FUNCTION Convert_BOOL_TO_LINT : Hresult
VAR_INPUT
	in : BOOL;
	out : REFERENCE TO LINT;
END_VAR
VAR
	converted : LINT;
END_VAR

converted := BOOL_TO_LINT(in);

IF (LINT_TO_BOOL(converted) <> in) THEN
	Convert_BOOL_TO_LINT := INCOMPATIBLE;
	RETURN;
END_IF

out := converted;

END_FUNCTION

(* stored: Version 1.1.0.1, ProductVersion 3.1.4024.12
   POU Convert_BOOL_TO_LINT: Id {c161c42b-6e14-4906-a7b9-f32aeb745424}, SpecialFunc None *)
